// TIA Portal V18 export
FUNCTION_BLOCK "vciLibBL"   // FB18, LAD
{ S7_Optimized_Access := 'TRUE' }
VERSION : 0.1
// stored: AutoNumber true, IsIECCheckEnabled false, IsRetainMemResEnabled false, MemoryReserve 100, SetENOAutomatically false, UDAEnableTagReadback false
   VAR_INPUT
      inBL01 : Int;
   END_VAR
   VAR_OUTPUT
      outBL01 : Real;
   END_VAR
   VAR_IN_OUT
      data : "udtBL";
   END_VAR
BEGIN

REGION Network 1: BL
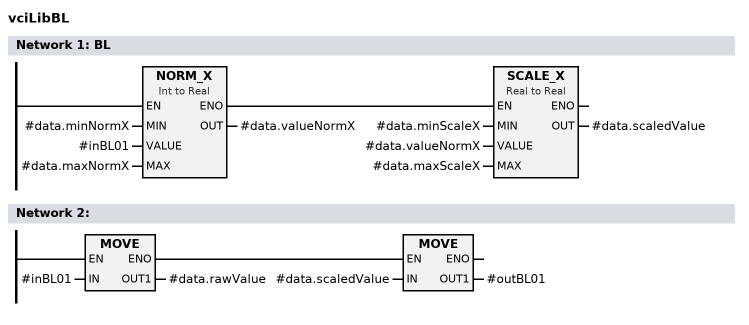
   RUNG wire#powerrail
      { S7_Templates := "[SrcType := Int, DestType := Real]"; S7_GenerateENO := "TRUE" } Normalize(min := #data.minNormX, value := #inBL01, max := #data.maxNormX, out => #data.valueNormX)
      { S7_Templates := "[SrcType := Real, DestType := Real]"; S7_GenerateENO := "TRUE" } Scale(min := #data.minScaleX, value := #data.valueNormX, max := #data.maxScaleX, out => #data.scaledValue)
   END_RUNG
   // the same network as SCL:
   // ENO of a box is taken as its EN; it also drops when the box reports an error
   #data.valueNormX := NORM_X(MIN := #data.minNormX, VALUE := #inBL01, MAX := #data.maxNormX);
   #data.scaledValue := SCALE_X(MIN := #data.minScaleX, VALUE := #data.valueNormX, MAX := #data.maxScaleX);
END_REGION

REGION Network 2
   RUNG wire#powerrail
      { S7_GenerateENO := "TRUE" } Move(in := #inBL01, out1 => #data.rawValue)
      { S7_GenerateENO := "TRUE" } Move(in := #data.scaledValue, out1 => #outBL01)
   END_RUNG
   // the same network as SCL:
   // ENO of a box is taken as its EN; it also drops when the box reports an error
   #data.rawValue := #inBL01;
   #outBL01 := #data.scaledValue;
END_REGION
END_FUNCTION_BLOCK
